DATA_BLOCK "TRANSPORTADORES_DB"
{ S7_Optimized_Access := 'TRUE' }
VERSION : 0.1
NON_RETAIN
"TRANSPORTADORES"

BEGIN

END_DATA_BLOCK

